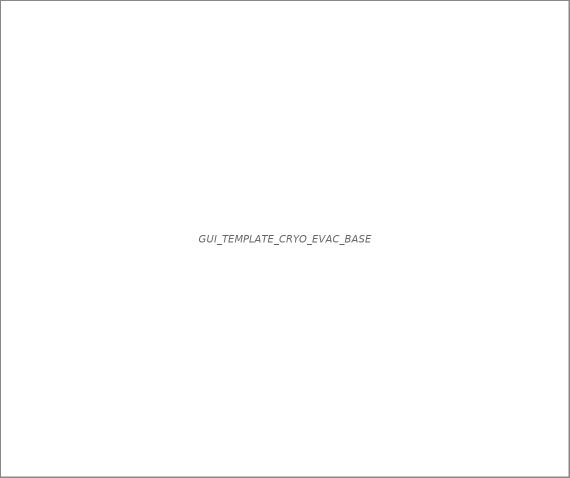
VISUALIZATION GUI_EVAC_LAB  // 570x478
    Frame (0,0 570x478)
        shows GUI_TEMPLATE_CRYO_EVAC_BASE(m_Instance := MAIN.evac_lab, m_bEnable := MAIN.bEnable_evac_lab)
END_VISUALIZATION

(* stored: Version 1.1.0.1, ProductVersion 3.1.4024.9
   Visu GUI_EVAC_LAB: Id {69381f5f-5b90-43a4-90ac-aa8800423257} *)
